{attribute 'qualified_only'}
TYPE Dialog_FormatTypes :
(
	DECIMAL := 0,
	HEX
);
END_TYPE

(* stored: Version 1.1.0.1, ProductVersion 3.1.4024.2
   DUT Dialog_FormatTypes: Id {7fe538e7-cb17-457b-b7da-fdd8cd1c0fe1} *)
